// TIA Portal V19 export
TYPE "LUC_typeModeRequests"
TITLE = LUC_typeStateModeManagerModes
// Unit Mode requests
// stored: Access Published
   STRUCT
      production : Bool := false;   // Request to change to "Production"
      maintenance : Bool := false;   // Request to change to "Maintenance"
      manual : Bool := false;   // Request to change to "Manual"
      userMode01 : Bool := false;   // Request to change to "UserMode01"
      userMode02 : Bool := false;   // Request to change to "UserMode02"
      userMode03 : Bool := false;   // Request to change to "UserMode03"
      userMode04 : Bool := false;   // Request to change to "UserMode04"
      userMode05 : Bool := false;   // Request to change to "UserMode05"
      userMode06 : Bool := false;   // Request to change to "UserMode06"
      userMode07 : Bool := false;   // Request to change to "UserMode07"
      userMode08 : Bool := false;   // Request to change to "UserMode8"
      userMode09 : Bool := false;   // Request to change to "UserMode9"
      userMode10 : Bool := false;   // Request to change to "UserMode10"
      userMode11 : Bool := false;   // Request to change to "UserMode11"
      userMode12 : Bool := false;   // Request to change to "UserMode12"
      userMode13 : Bool := false;   // Request to change to "UserMode13"
   END_STRUCT;
END_TYPE
